Staubli VAL3: programList.pgx

program programList(string& x_sEvent[])
  local num nSize
  local string sEvent
  local num lKey
  local num i
  local string message
begin
  //
  // USE this procedure to view Prog
  // that you have already saved
  //
  cls()
  call use:setView(false)
  //
  // Prog
  //
  call use:listcreate("PROG ")
  //
  call prog:getSize(nSize)
  // refresh the list
  for i=0 to nSize-1
    call prog:get(sEvent,i)
    if sEvent!="" and find(sEvent,"#")==-1 and sEvent!="HOME1" and sEvent!="HOME2"
      call use:listadd(sEvent)
    endIf
  endFor
  call use:listupdate(0)
  call language:message(message,60)
  call use:typeLen(0,13,message,40)
  do
    lKey=get()
    call use:listevent(lKey,i,x_sEvent)
  until lKey==270 or lKey==255
  if lKey==255
    x_sEvent=""
  endIf
end
